FUNCTION RandomizeArray
VAR
	lower: DINT;
	upper: DINT;
	i: DINT;

END_VAR
VAR_IN_OUT
	target: ARRAY[*] OF LREAL;
END_VAR

lower := LOWER_BOUND(target, 1);
upper := UPPER_BOUND(target, 1);

FOR i:=lower TO upper DO
  GVL.rand_generator(Num=>target[i]);
END_FOR

END_FUNCTION

(* stored: Version 1.1.0.1, ProductVersion 3.1.4026.0
   POU RandomizeArray: Id {37f861ee-38e4-40f2-af01-7e9beb004c5f}, SpecialFunc None *)
